# EPICS substitutions: iocs/xspress3IOC/iocBoot/iocXspress3/xsp3-4ch.substitutions
file "$(ADXSPRESS3)/db/xspress3Channel.db"
{
pattern { P, R, PORT, ADDR, CHAN, TIMEOUT }
{ "$(P_)", "", "$(PORT_)", 0, 1, 1 }
{ "$(P_)", "", "$(PORT_)", 1, 2, 1 }
{ "$(P_)", "", "$(PORT_)", 2, 3, 1 }
{ "$(P_)", "", "$(PORT_)", 3, 4, 1 }
}
